FUNCTION_BLOCK FIELDBUS_UINT_TO_SIGNAL_COMPOUND_SCALE (* Mirrors IN->OUT if Signal Valid, with compound scaling for upper and lower byte *)
  (* Standard: 61499-1; Description: Copyright (c) 2026 HR Agrartechnik GmbH This program and the accompanying materials are made available under the terms of the Eclipse Public License 2.0 which is available at https://www.eclipse.org/legal/epl-2.0/ SPDX-License-Identifier: EPL-2.0 *)
  (* Version 1.0, 2026-05-31, Franz Höpfinger, HR Agrartechnik GmbH *)
  PACKAGE logiBUS::signalprocessing::fieldbus;
  IMPORT eclipse4diac::signalprocessing::FIELDBUS_SIGNAL::NOT_AVAILABLE_WM;
  IMPORT eclipse4diac::signalprocessing::FIELDBUS_SIGNAL::VALID_SIGNAL_W;
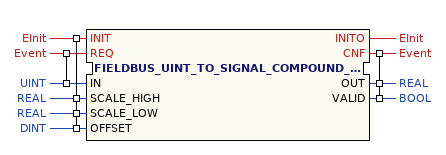
  EVENT_INPUT
    INIT : EInit WITH SCALE_HIGH, SCALE_LOW, OFFSET; (* Init Request *)
    REQ WITH IN; (* Normal Execution Request *)
  END_EVENT
  EVENT_OUTPUT
    INITO : EInit; (* Init Confirmation *)
    CNF WITH OUT, VALID; (* Execution Confirmation *)
  END_EVENT
  VAR_INPUT
    IN : UINT := WORD_TO_UINT(NOT_AVAILABLE_WM); (* Input *)
    SCALE_HIGH : REAL := REAL#0.256; (* Scale factor for upper byte *)
    SCALE_LOW : REAL := REAL#0.001; (* Scale factor for lower byte *)
    OFFSET : DINT := DINT#0; (* Offset added after scaling *)
  END_VAR
  VAR_OUTPUT
    OUT : REAL := REAL#0.0; (* Output Scaled *)
    VALID : BOOL := FALSE; (* TRUE if Signal is VALID *)
  END_VAR
  VAR
    temp : WORD;
    highByte : WORD;
    lowByte : WORD;
  END_VAR
  EC_STATES
    INIT : INIT -> INITO;
    REQ : REQ -> CNF;
  END_STATES
  ALGORITHM INIT IN ST:

  END_ALGORITHM
  ALGORITHM REQ IN ST: (* Executed algorithm *)
IF (IN <= WORD_TO_UINT(VALID_SIGNAL_W)) THEN
	temp := SHR(UINT_TO_WORD(IN), SINT#8);
	highByte := temp AND WORD#16#00FF;
	lowByte := UINT_TO_WORD(IN) AND WORD#16#00FF;
	OUT := UINT_TO_REAL(WORD_TO_UINT(highByte)) * SCALE_HIGH + UINT_TO_REAL(WORD_TO_UINT(lowByte)) * SCALE_LOW
		+ DINT_TO_REAL(OFFSET);
	VALID := BOOL#TRUE;
ELSE
	OUT := REAL#0.0;
	VALID := BOOL#FALSE;
END_IF;
  END_ALGORITHM
END_FUNCTION_BLOCK
